{attribute 'qualified_only'}
VAR_GLOBAL
	fbSterowanieMaszyna						: FB_SterowanieMaszyna;
	
END_VAR

(* stored: Version 1.1.0.1, ProductVersion 3.1.4024.11
   GVL GVL_SterowanieMaszyna: Id {0eff2586-3070-474c-a58f-f57dff475ef9} *)
